INTERFACE I_CollectionChangedEvent EXTENDS I_Event

PROPERTY PUBLIC Target : I_Collection
GET
END_GET
END_PROPERTY

END_INTERFACE

(* stored: Version 1.1.0.1, ProductVersion 3.1.4024.12
   Itf I_CollectionChangedEvent: Id {4d9aaefe-74aa-0c75-3e3c-563b94981f7b}
   Property Target: Id {c58e6b87-594b-093a-34b0-80bd61141f42}
   Get Get: Id {2ddcbc65-b8f7-005b-227a-6551b371da0d} *)
